// Mitsubishi GX Works2 project: a19   PLC: Q02/Q02H

PROGRAM MAIN
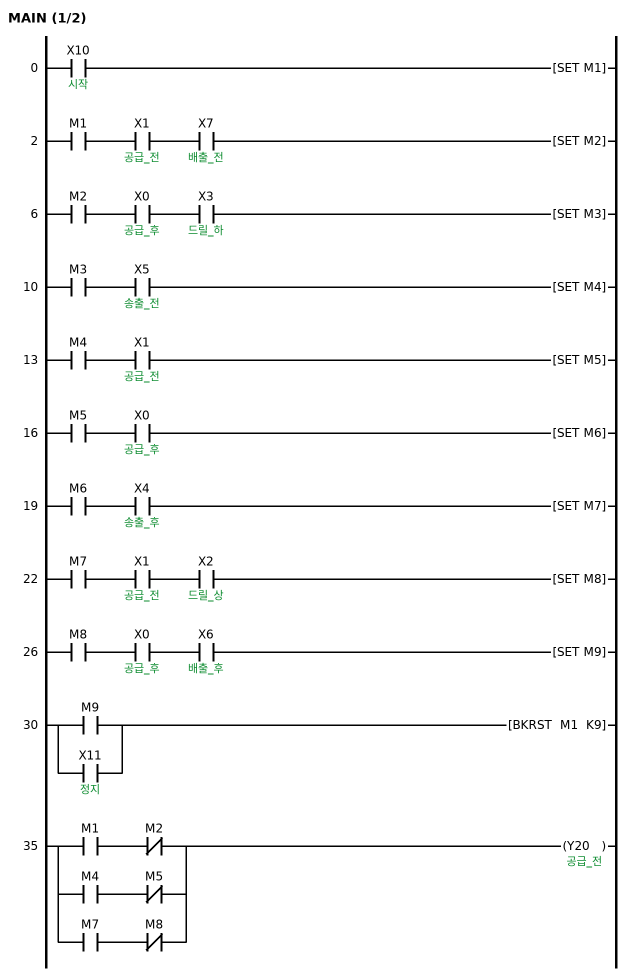
0     LD      X10  ; 시작
      SET     M1
2     LD      M1
      AND     X1  ; 공급_전
      AND     X7  ; 배출_전
      SET     M2
6     LD      M2
      AND     X0  ; 공급_후
      AND     X3  ; 드릴_하
      SET     M3
10    LD      M3
      AND     X5  ; 송출_전
      SET     M4
13    LD      M4
      AND     X1  ; 공급_전
      SET     M5
16    LD      M5
      AND     X0  ; 공급_후
      SET     M6
19    LD      M6
      AND     X4  ; 송출_후
      SET     M7
22    LD      M7
      AND     X1  ; 공급_전
      AND     X2  ; 드릴_상
      SET     M8
26    LD      M8
      AND     X0  ; 공급_후
      AND     X6  ; 배출_후
      SET     M9
30    LD      M9
      OR      X11  ; 정지
      BKRST   M1 K9
35    LD      M1
      ANI     M2
      LD      M4
      ANI     M5
      ORB
      LD      M7
      ANI     M8
      ORB
      OUT     Y20  ; 공급_전
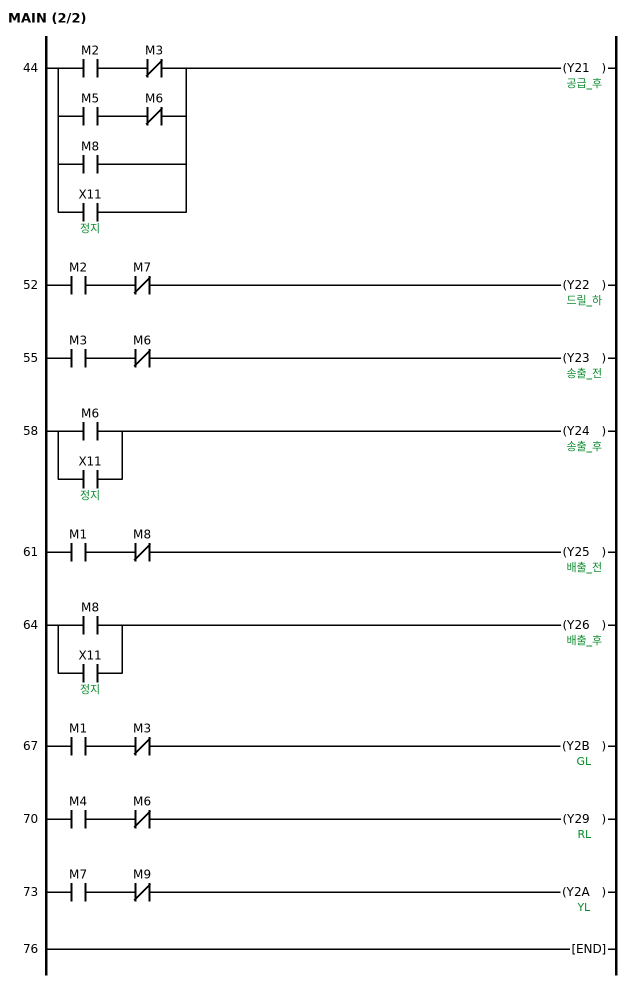
44    LD      M2
      ANI     M3
      LD      M5
      ANI     M6
      ORB
      OR      M8
      OR      X11  ; 정지
      OUT     Y21  ; 공급_후
52    LD      M2
      ANI     M7
      OUT     Y22  ; 드릴_하
55    LD      M3
      ANI     M6
      OUT     Y23  ; 송출_전
58    LD      M6
      OR      X11  ; 정지
      OUT     Y24  ; 송출_후
61    LD      M1
      ANI     M8
      OUT     Y25  ; 배출_전
64    LD      M8
      OR      X11  ; 정지
      OUT     Y26  ; 배출_후
67    LD      M1
      ANI     M3
      OUT     Y2B  ; GL
70    LD      M4
      ANI     M6
      OUT     Y29  ; RL
73    LD      M7
      ANI     M9
      OUT     Y2A  ; YL
76    END
END_PROGRAM
